{attribute 'GeneratedUsingTerminal: EL5001-0011-0016'}
{attribute addProperty BoxType "EL5001-0011-0016"}
{attribute addProperty Id "SSI_InputsAT %I*SSI_Inputs_3B70A31110WcStateAT %I*WcState_9091E0EB2InfoDataAT %I*InfoData_1088C70510"}
{attribute addProperty CRC "1878436041"}
{attribute addProperty Size "22"}
TYPE EL5001_6FF6A8C9 EXTENDS EtcSlaveTerminalBase_947E5A46 :
STRUCT
	{attribute addProperty Name "SSI_Inputs"}
	SSI_Inputs : SSI_Inputs_3B70A311;
	{attribute addProperty Name "WcState"}
	WcState : WcState_9091E0EB;
	{attribute addProperty Name "InfoData"}
	InfoData : InfoData_1088C705;
END_STRUCT
END_TYPE

(* stored: Version 1.2.0.0, ProductVersion 3.1.4024.9
   DUT EL5001_6FF6A8C9: Id {fd0da75b-e1f4-4833-b573-9d327eef7413} *)
